FUNCTION_BLOCK ABSTRACT FB_PMLModuleBase IMPLEMENTS ITF_PMLModuleBase
VAR CONSTANT
	//Constant declarations
	PRODUCTION_DATA_ALARM_COUNT	: UDINT := 16;
END_VAR
VAR PERSISTENT
	//ITF_ProductionData internal variables
	tShiftLength: TIME := T#10M;
	nShiftProductionTarget	: DINT := 1000;
	fWarningMargin			: LREAL := 10;
	fProductionRate_Setpoint	: LREAL := 30;
	nRateAveragingCount		: DINT := 10;
END_VAR
VAR
	//ITF_PMLModuleBase internal property variables
	sAncestorIDs		: STRING;				//String concatenation of preceding parent IDs to prefix this module's ID
	bLogModeChanges 	: BOOL := TRUE; 		//Toggle to permit or suppress state change logging (Should be tied to HMI setting to optionally reduce event logger clutter)
	bLogStateChanges 	: BOOL := FALSE; 		//Toggle to permit or suppress state change logging (Should be tied to HMI setting to optionally reduce event logger clutter)
	nModuleID			: UDINT;					//Unique identifying number for the module
	sModuleName			: STRING;				//Human-readable module name for user-side messaging
	bEnabled			: BOOL := TRUE;			//Enables or disables the packml Machine of the module (prevents the module from going past idle)
	eModeCommand		: E_PMLUnitMode; 				//Current Commanded UnitMode of the module
	eStateCommand		: Tc3_PackML_V2.E_PMLCommand;
	eMode				: E_PMLUnitMode;		//Current UnitMode of the module
	eState				: Tc3_PackML_V2.E_PMLState;
	iMasterDataStructure_Adder : ITF_Tree_IndexBased;
	eCurrentAlarmSeverity		: TcEventSeverity;
	a_eParentFaultResponseDefinitions		: ARRAY[0..4] OF E_AlarmResponse := [	E_AlarmResponse.NoResponse,
																					E_AlarmResponse.NoResponse,
																					E_AlarmResponse.NoResponse,
																					E_AlarmResponse.Abort_ImmediateError,
																					E_AlarmResponse.Abort_ImmediateError];
	
	fbFIFO							: FB_FIFO_ULINT_Array;
	a_fbProductionDataAlarms		: ARRAY[1..PRODUCTION_DATA_ALARM_COUNT] OF FB_TcAlarm;
	fTemp : LREAL;



	//Communication Variables
	stPMLModuleBaseHMI	: ST_PMLModuleBase_HMI;		//Handles status and control communications with the HMI
	stPMLModuleBaseVISU	: ST_PMLModuleBase_VISU;	//Handles status and control communications with Visualizations
	fbExternalControl	: FB_ModuleExternalCommandControl;	//Handles commands from HMI/VISUS ^^ kind of overlaps with the structures above - TODO: Improve

	//Administration and Configuration Variables
	bInitialized 					: BOOL;					//TRUE when initialization code of the object is complete
	sID_Name						: STRING;				//"Module XX - 'Module Name' " Alarm and message utility phrase based off of nMachine ID and sMachineName
	
	//State and Mode control blocks
	fbModeManager 					: PML_UnitModeManager; 	//Manages operating mode transitions and rules
	fbStateMachine 					: PML_StateMachine; 	//Manages PackML state transitions
	fbCustomModes 					: PML_UnitModeConfig;	//Used to define custom machine modes if desired

	//State and Mode Status and Command variables
	sState							: STRING; 				//String representation of the current state
	eLastState						: E_PMLState;			//Last cycle PackML state
	eLastStateCommand				: E_PMLCommand;			//Previous received PackML state command
	eLastMode		 				: DINT;					//Last PackML mode 
	eLastModeCommand 				: E_PMLUnitMode;					//Previous received PackML mode command
	bStateTasksComplete				: BOOL := FALSE;					//All tasks to be performed at this program level are complete
	bNoStateTasksToComplete			: BOOL := TRUE;					//Indicates whether this stateneeds to perform tasks other than commanding its children
	bSubModulesReady				: BOOL;					//All submodules have reached the commanded state
	
	//Alarming and Logging variables - Some may or may not be necessary depending on final alarm system implementation ----------------------------------------------
	//These are for the newer TMC Excel import style alarm system
	a_fbPMLAlarms					: ARRAY[1..48] OF FB_TcAlarm;	//Array of alarms for PackML state and mode changes that exist in any PackML enabled module
	a_fbBaseAlarms					: ARRAY[1..32] OF FB_TcAlarm;		//Array of alarms for general module Alarms				
	fbPMLStateLogger				: FB_PMLStateLogger;				//Logs PackML state changes
	fbPMLModeLogger					: FB_PMLModeLogger;					//Logs PackML Mode changes

	// Alarm handling
	bActiveAlarm					: BOOL;					//module has an active alarm		TODO: Implement			
	bGlobalSafetyStatus				: BOOL;
	//********************************************************************************************************************
	// Sub Module variables
	// Used mostly for EMs and Machines, but ok for CM. They are just null	
	a_ITF_PackMLBase				: ARRAY[1..MAX_NO_OF_SUBMODULES] OF ITF_PMLModuleBase;	
	// Array of the PML sub unit info array used by the statemachine
	a_stPMLSubUnitInfo				: ARRAY[1..MAX_NO_OF_SUBMODULES] OF ST_PMLSubUnitInfo;
	nNumberOfSubModules				: UDINT := 0;	//calculated number of instantiated sub modules
	// This is the information for each module's submodules.
	PMLSubUnitInfoRef				: ST_PMLSubUnitInfoRef;				// Reference to the subunit information, used by the state machine
	//********************************************************************************************************************
	
	//Component variables - Allow iterative control of child components (Mostly used with Control Modules, but usable anywhere)
	a_ITF_Components				: ARRAY[1..MAX_NO_OF_COMPONENTS] OF ITF_ComponentBase;
	nNumberOfComponents				: UDINT := 0;	//calculated number of instantiated components
	
	//Miscellaneous Variables
	fLastProductionRate_Setpoint 	: LREAL;
	nIndex							: UDINT;		//Generic iteration value
	bSimulateAllChildren			: BOOL;
	a_sModeNames					: ARRAY[0..31] OF STRING;
	varInfo							: __SYSTEM.VAR_INFO;
	bReachedInitialDefaultStateAndMode	: BOOL;		//Toggles TRUE once a module has reached the default state and mode after startup, used to mute certain alarms during startup
	i: UDINT;
END_VAR

//*********************************************************
// !!!!! Code implementation only in CyclicLogic() method !!!!! 
//*********************************************************

METHOD Aborted
//*************************************************************************************************************************************************************************
//If you are about to write application specific code, note that any such code should exist within the "Application" directory using a Function Block that 'EXTENDS' this base Function Block!
//This particular method's functionality can be overriden in the extended block by creating a method of the same name, with desired functionality therein
//If the functionality of this base module is to be retained, but more functionality is desired, the extended method can contain a SUPER^.ThisMethodName(); call, which will call this code
//*************************************************************************************************************************************************************************

;
END_METHOD

METHOD AbortImmediate : BOOL
VAR_INPUT
END_VAR
eStateCommand := E_PMLCommand.ePMLCommand_Abort;
END_METHOD

METHOD AbortImmediateError : BOOL
VAR_INPUT
	sName		: STRING;
	bIsModule	: BOOL;
END_VAR
IF bIsModule THEN
	IF NOT a_fbBaseAlarms[E_BaseAlarms.SubModuleError].bRaised THEN
		F_RaiseAlarmWithStringParameters(a_fbBaseAlarms[E_BaseAlarms.SubModuleError],sModuleName,sName,'');
	END_IF
ELSE
	IF NOT a_fbBaseAlarms[E_BaseAlarms.ComponentError].bRaised THEN
		F_RaiseAlarmWithStringParameters(a_fbBaseAlarms[E_BaseAlarms.ComponentError],sModuleName,sName,'');
	END_IF
END_IF


eStateCommand := E_PMLCommand.ePMLCommand_Abort;
END_METHOD

METHOD Aborting
//*************************************************************************************************************************************************************************
//If you are about to write application specific code, note that any such code should exist within the "Application" directory using a Function Block that 'EXTENDS' this base Function Block!
//This particular method's functionality can be overriden in the extended block by creating a method of the same name, with desired functionality therein
//If the functionality of this base module is to be retained, but more functionality is desired, the extended method can contain a SUPER^.ThisMethodName(); call, which will call this code
//*************************************************************************************************************************************************************************

//Perform State tasks here
// Send abort command to all sub modules
FOR nIndex := 1 TO nNumberOfSubModules DO
	a_ITF_PackMLBase[nIndex].StateCommand:=ePMLCommand_Abort;
END_FOR

// All subunits in requested state?
bSubModulesReady := TRUE;

FOR nIndex := 1 TO nNumberOfSubModules DO
	bSubModulesReady := bSubModulesReady AND (a_ITF_PackMLBase[nIndex].State = ePMLState_Aborted);
END_FOR
IF bSubModulesReady AND (bStateTasksComplete OR bNoStateTasksToComplete) THEN
	bNoStateTasksToComplete := TRUE;
	bStateTasksComplete := FALSE;
	StateComplete();
END_IF
END_METHOD

METHOD AllowHMIControl : BOOL
VAR_INPUT
	bModuleOnly		: BOOL;	//If TRUE, only the PML module itself is controllable, If FALSE, all components become controllable as well
END_VAR
stPMLModuleBaseHMI.bHMIControlAvailable := TRUE;

IF bModuleOnly THEN
	FOR i := 1 TO nNumberOfComponents DO
		a_ITF_Components[i].BlockHMIControl();
	END_FOR
ELSE
	FOR i := 1 TO nNumberOfComponents DO
		a_ITF_Components[i].AllowHMIControl();
	END_FOR
END_IF
END_METHOD

PROPERTY AncestorIDs : STRING
GET
AncestorIDs := sAncestorIDs;
END_GET
SET
sAncestorIDs := AncestorIDs;
END_SET
END_PROPERTY

METHOD BlockHMIControl : BOOL
VAR_INPUT
END_VAR
stPMLModuleBaseHMI.bHMIControlAvailable := FALSE;

FOR i := 1 TO nNumberOfComponents DO
	a_ITF_Components[i].BlockHMIControl();
END_FOR
END_METHOD

METHOD Clearing
//*************************************************************************************************************************************************************************
//If you are about to write application specific code, note that any such code should exist within the "Application" directory using a Function Block that 'EXTENDS' this base Function Block!
//This particular method's functionality can be overriden in the extended block by creating a method of the same name, with desired functionality therein
//If the functionality of this base module is to be retained, but more functionality is desired, the extended method can contain a SUPER^.ThisMethodName(); call, which will call this code
//*************************************************************************************************************************************************************************

//Perform State tasks here
// Send clear command to all sub modules
FOR nIndex := 1 TO nNumberOfSubModules DO	
	a_ITF_PackMLBase[nIndex].StateCommand := ePMLCommand_Clear;
END_FOR

IF a_fbBaseAlarms[E_BaseAlarms.ComponentError].bRaised THEN
	a_fbBaseAlarms[E_BaseAlarms.ComponentError].Clear(0,0);
END_IF;

IF a_fbBaseAlarms[E_BaseAlarms.SubModuleError].bRaised THEN
	a_fbBaseAlarms[E_BaseAlarms.SubModuleError].Clear(0,0);
END_IF;


// All subunits in requested state?
bSubModulesReady	:= TRUE;
FOR nIndex:=1 TO nNumberOfComponents DO
	IF a_ITF_Components[nIndex].Error THEN
		a_ITF_Components[nIndex].Reset();
	END_IF
END_FOR

FOR nIndex:=1 TO nNumberOfComponents DO		
		bSubModulesReady := bSubModulesReady AND NOT a_ITF_Components[nIndex].Error;
END_FOR

FOR nIndex := 1 TO nNumberOfSubModules DO
	bSubModulesReady := bSubModulesReady AND (a_ITF_PackMLBase[nIndex].State = ePMLState_Stopped);
END_FOR
IF bSubModulesReady AND (bStateTasksComplete OR bNoStateTasksToComplete) THEN
	bNoStateTasksToComplete := TRUE;
	bStateTasksComplete := FALSE;
	StateComplete();
END_IF
END_METHOD

METHOD Complete
//*************************************************************************************************************************************************************************
//If you are about to write application specific code, note that any such code should exist within the "Application" directory using a Function Block that 'EXTENDS' this base Function Block!
//This particular method's functionality can be overriden in the extended block by creating a method of the same name, with desired functionality therein
//If the functionality of this base module is to be retained, but more functionality is desired, the extended method can contain a SUPER^.ThisMethodName(); call, which will call this code
//*************************************************************************************************************************************************************************

;
END_METHOD

METHOD Completing
//*************************************************************************************************************************************************************************
//If you are about to write application specific code, note that any such code should exist within the "Application" directory using a Function Block that 'EXTENDS' this base Function Block!
//This particular method's functionality can be overriden in the extended block by creating a method of the same name, with desired functionality therein
//If the functionality of this base module is to be retained, but more functionality is desired, the extended method can contain a SUPER^.ThisMethodName(); call, which will call this code
//*************************************************************************************************************************************************************************

//Perform State tasks here
// Send complete command to all sub modules
FOR nIndex := 1 TO nNumberOfSubModules DO
	a_ITF_PackMLBase[nIndex].StateCommand:=ePMLCommand_Complete;
END_FOR

// All subunits in requested state?
bSubModulesReady	:= TRUE;
FOR nIndex := 1 TO nNumberOfSubModules DO
	bSubModulesReady := bSubModulesReady AND (a_ITF_PackMLBase[nIndex].State = ePMLState_Complete);
END_FOR
IF bSubModulesReady AND (bStateTasksComplete OR bNoStateTasksToComplete) THEN
	bNoStateTasksToComplete := TRUE;
	bStateTasksComplete := FALSE;
	StateComplete();
END_IF
END_METHOD

METHOD ComponentMonitor : BOOL
VAR
	a_eAlarmResponses		: ARRAY[0..4] OF E_AlarmResponse;	//Temporary response array
END_VAR
FOR i:=1 TO nNumberOfComponents DO
	IF bSimulateAllChildren THEN
		a_ITF_Components[i].Simulate := TRUE;
	ELSE 
		a_ITF_Components[i].Simulate := FALSE;
	END_IF
	
	IF eMode = E_PMLUnitMode.ePMLUnitMode_Production THEN
		IF 		eState <> E_PMLState.ePMLState_Aborted
			AND eState <> E_PMLState.ePMLState_Aborting
			AND eState <> E_PMLState.ePMLState_Clearing
			AND eState <> E_PMLState.ePMLState_Stopped
			AND eState <> E_PMLState.ePMLState_Stopping
		THEN
			a_eAlarmResponses := a_ITF_Components[i].ParentResponseDefinitions;
			CASE a_eAlarmResponses[a_ITF_Components[i].CurrentAlarmSeverity] OF
				E_AlarmResponse.Abort_ImmediateError:
					AbortImmediateError(a_ITF_Components[i].Name, FALSE);
				E_AlarmResponse.Abort_Immediate:
					AbortImmediate();
				E_AlarmResponse.Stop_Immediate:
					StopImmediate();
				E_AlarmResponse.Stop_Controlled:
					StopControlled();
				E_AlarmResponse.Hold_Immediate:
					HoldImmediate();
				E_AlarmResponse.Suspend_Immediate:
					SuspendImmediate();
				E_AlarmResponse.Suspend_Controlled:
					SuspendControlled();
				E_AlarmResponse.NoResponse:
					;
			END_CASE
		ELSIF eState = E_PMLState.ePMLState_Stopped
			OR eState = E_PMLState.ePMLState_Stopping 
		THEN
			a_eAlarmResponses := a_ITF_Components[i].ParentResponseDefinitions;
			CASE a_eAlarmResponses[a_ITF_Components[i].CurrentAlarmSeverity] OF
				E_AlarmResponse.Abort_ImmediateError:
					AbortImmediateError(a_ITF_Components[i].Name, FALSE);
				E_AlarmResponse.Abort_Immediate:
					AbortImmediate();
				E_AlarmResponse.NoResponse:
					;
			END_CASE				
		END_IF
	END_IF		
END_FOR
END_METHOD

{attribute 'call_after_online_change_slot' := '<slot>'}
METHOD CreateEvents : BOOL
VAR_INPUT
END_VAR

VAR
END_VAR

F_CreateAllEventsInClass(	p_aAlarms := a_fbPMLAlarms,
							nClassSize := SIZEOF(TC_EVENTS.PMLAlarms),
							pInitEvent := ADR(TC_EVENTS.PMLAlarms.InitReferenceEvent),
							sPrefix := sID_Name);
							
F_CreateAllEventsInClass(	p_aAlarms := a_fbBaseAlarms,
							nClassSize := SIZEOF(TC_EVENTS.BaseAlarms),
							pInitEvent := ADR(TC_EVENTS.BaseAlarms.InitReferenceEvent),
							sPrefix := sID_Name);							
							
F_CreateAllEventsInClass(	p_aAlarms := a_fbProductionDataAlarms,
							nClassSize := SIZEOF(TC_EVENTS.ProductionData),
							pInitEvent := ADR(TC_EVENTS.ProductionData.InitReferenceEvent),
							sPrefix := sID_Name);
END_METHOD

PROPERTY CurrentAlarmSeverity : TcEventSeverity
GET
CurrentAlarmSeverity := eCurrentAlarmSeverity;
END_GET
END_PROPERTY

// 
// Cyclic Code
METHOD CyclicLogic
//*********************************************************
//If you are about to write actual machine implementation code, note that implementation code should exist within an implementation machine module block that extends this machine module base!
//*********************************************************

// First loop initialization code is triggered by highest level class
IF NOT bInitialized THEN			//Force initialization code of the object
	initialize();
	bInitialized := TRUE;
END_IF

//TODO: Condition state based on DEFAULT constant, right now it is a command, so a case statement translation to state would be necessary
IF NOT bReachedInitialDefaultStateAndMode AND eState = E_PMLState.ePMLState_Aborted AND eMode = ePMLUNITMODEDEFAULT THEN
	bReachedInitialDefaultStateAndMode := TRUE;
END_IF

//  call the subunits
FOR i := 1 TO nNumberOfSubModules DO	
	a_ITF_PackMLBase[i].CyclicLogic();								//Call the main cyclic loop of the subunits 
	a_stPMLSubUnitInfo[i].eState := a_ITF_PackMLBase[i].State;  	//Reflect the state of the subunits to the state machine of the module
END_FOR

FOR i:=1 TO nNumberOfComponents DO
	IF a_ITF_Components[i] <> 0 THEN
		a_ITF_Components[i].CyclicLogic();
	END_IF
END_FOR


// Mode control loop of the module
ModeControl();

// State control loop of the module
StateControl();

HMICommunication();
VISUCommunication();
fbExternalControl();
SubModuleMonitor();
ComponentMonitor();
HMIPermissions();

eCurrentAlarmSeverity := TcEventSeverity.Verbose;

eCurrentAlarmSeverity := F_GetMaxSeverityRaised(	a_fbAlarms := a_fbPMLAlarms,
													eCurrentSeverity := eCurrentAlarmSeverity);
eCurrentAlarmSeverity := F_GetMaxSeverityRaised(	a_fbAlarms := a_fbBaseAlarms,
													eCurrentSeverity := eCurrentAlarmSeverity);
END_METHOD

PROPERTY Enabled : BOOL
GET
Enabled := bEnabled;
END_GET
SET
bEnabled := Enabled;
END_SET
END_PROPERTY

METHOD Execute
//*************************************************************************************************************************************************************************
//If you are about to write application specific code, note that any such code should exist within the "Application" directory using a Function Block that 'EXTENDS' this base Function Block!
//This particular method's functionality can be overriden in the extended block by creating a method of the same name, with desired functionality therein
//If the functionality of this base module is to be retained, but more functionality is desired, the extended method can contain a SUPER^.ThisMethodName(); call, which will call this code
//*************************************************************************************************************************************************************************

;
END_METHOD

METHOD Held
//*************************************************************************************************************************************************************************
//If you are about to write application specific code, note that any such code should exist within the "Application" directory using a Function Block that 'EXTENDS' this base Function Block!
//This particular method's functionality can be overriden in the extended block by creating a method of the same name, with desired functionality therein
//If the functionality of this base module is to be retained, but more functionality is desired, the extended method can contain a SUPER^.ThisMethodName(); call, which will call this code
//*************************************************************************************************************************************************************************
END_METHOD

METHOD HMICommunication : BOOL
//Extend this method in extended FBs to communicate specific implementation data

//Process HMI requests
IF stPMLModuleBaseHMI.bIncomingHMIRequest AND NOT stPMLModuleBaseHMI.bHMICommandConfirmation THEN		//If a request has been issued by the HMI, and a previous request has not just E_SequenceState.Finished being processed
	
	IF stPMLModuleBaseHMI.bHMIControlAvailable THEN		//If the current conditions permit HMI control (Should be determined by the extended application components)
		IF stPMLModuleBaseHMI.bEnableHMIRequest THEN
			bEnabled := TRUE;
			stPMLModuleBaseHMI.bHMICommandConfirmation := TRUE;	//Confirm that the request has been processed
		END_IF
		IF stPMLModuleBaseHMI.bDisableHMIRequest THEN
			bEnabled := FALSE;
			stPMLModuleBaseHMI.bHMICommandConfirmation := TRUE;	//Confirm that the request has been processed
		END_IF
		IF stPMLModuleBaseHMI.bStateCommandHMIRequest THEN
			eStateCommand := stPMLModuleBaseHMI.eStateCommandHMIValue;
			//fbExternalControl.ExternalControlHMI.StateCommand := stPMLModuleBaseHMI.eStateCommandHMIValue;
			//fbExternalControl.ExternalControlHMI.StateCommandPulse := TRUE;
			stPMLModuleBaseHMI.bHMICommandConfirmation := TRUE;	//Confirm that the request has been processed
		END_IF
		IF stPMLModuleBaseHMI.bModeCommandHMIRequest THEN
			eModeCommand := stPMLModuleBaseHMI.eModeCommandHMIValue;
			//fbExternalControl.ExternalControlHMI.ModeCommand := stPMLModuleBaseHMI.eModeCommandHMIValue;
			//fbExternalControl.ExternalControlHMI.ModeCommandPulse := TRUE;
			stPMLModuleBaseHMI.bHMICommandConfirmation := TRUE;	//Confirm that the request has been processed
		END_IF
	END_IF
	
		//The following commands are always permissible, and are therefore not conditioned with bHMIControlAvailable
	IF stPMLModuleBaseHMI.bActivateStateLogHMIRequest THEN
		bLogStateChanges := TRUE;
		stPMLModuleBaseHMI.bHMICommandConfirmation := TRUE;	//Confirm that the request has been processed
	END_IF
	IF stPMLModuleBaseHMI.bDeactivateStateLogHMIRequest THEN
		bLogStateChanges := FALSE;
		stPMLModuleBaseHMI.bHMICommandConfirmation := TRUE;	//Confirm that the request has been processed
	END_IF
	IF stPMLModuleBaseHMI.bActivateModeLogHMIRequest THEN
		bLogModeChanges := TRUE;
		stPMLModuleBaseHMI.bHMICommandConfirmation := TRUE;	//Confirm that the request has been processed
	END_IF
	IF stPMLModuleBaseHMI.bDeactivateModeLogHMIRequest THEN
		bLogModeChanges := FALSE;
		stPMLModuleBaseHMI.bHMICommandConfirmation := TRUE;	//Confirm that the request has been processed
	END_IF		
END_IF


//Update HMI status info
stPMLModuleBaseHMI.bEnabled := bEnabled;
stPMLModuleBaseHMI.eMode := eMode;		//KAB eMode;
stPMLModuleBaseHMI.nModuleID := nModuleID;
stPMLModuleBaseHMI.sModuleName := sModuleName;
stPMLModuleBaseHMI.eState := eState;	//KAB eState;
stPMLModuleBaseHMI.bLogStateChanges := bLogStateChanges;
stPMLModuleBaseHMI.bLogModeChanges := bLogModeChanges;
stPMLModuleBaseHMI.a_sModeNames := a_sModeNames;
END_METHOD

PROPERTY HMIControlAvailable : BOOL
GET
HMIControlAvailable := stPMLModuleBaseHMI.bHMIControlAvailable;
END_GET
SET
stPMLModuleBaseHMI.bHMIControlAvailable := HMIControlAvailable;
END_SET
END_PROPERTY

METHOD HMIPermissions : BOOL
VAR_INPUT
END_VAR
//General Mode Based Monitoring and handling of HMI control
CASE eMode OF
//	====================================================================================================================================	
	E_PMLUnitMode.ePMLUnitMode_Production:			//=================================PRODUCTION MODE==================================
		CASE eState OF
			E_PMLState.ePMLState_Stopped:
				AllowHMIControl(bModuleOnly := TRUE);		//Allow control for recovery
			E_PMLState.ePMLState_Idle:
				BlockHMIControl();
			E_PMLState.ePMLState_Suspended:
				BlockHMIControl();
			E_PMLState.ePMLState_Execute:
				BlockHMIControl();
			E_PMLState.ePMLState_Aborted:
				AllowHMIControl(bModuleOnly := TRUE);		//Allow control for recovery
			E_PMLState.ePMLState_Held:
				AllowHMIControl(bModuleOnly := TRUE);		//Allow control for recovery
			E_PMLState.ePMLState_Complete:
				BlockHMIControl();
		END_CASE
		
//	====================================================================================================================================	
	E_PMLUnitMode.ePMLUnitMode_Manual:				//=================================MANUAL MODE======================================
		AllowHMIControl(bModuleOnly := FALSE);
//	====================================================================================================================================	
	E_PMLUnitMode.ePMLUnitMode_Maintenance:			//=================================MAINTENANCE MODE=================================
		AllowHMIControl(bModuleOnly := FALSE);	
END_CASE
END_METHOD

METHOD HoldControlled : BOOL
VAR_INPUT
END_VAR
END_METHOD

METHOD HoldImmediate : BOOL
VAR_INPUT
END_VAR
END_METHOD

METHOD Holding
//*************************************************************************************************************************************************************************
//If you are about to write application specific code, note that any such code should exist within the "Application" directory using a Function Block that 'EXTENDS' this base Function Block!
//This particular method's functionality can be overriden in the extended block by creating a method of the same name, with desired functionality therein
//If the functionality of this base module is to be retained, but more functionality is desired, the extended method can contain a SUPER^.ThisMethodName(); call, which will call this code
//*************************************************************************************************************************************************************************

//Perform State tasks here
// Send hold command to all sub modules
FOR nIndex := 1 TO nNumberOfSubModules DO
	a_ITF_PackMLBase[nIndex].StateCommand:=ePMLCommand_Hold;
END_FOR

// All subunits in requested state?
bSubModulesReady	:= TRUE;
FOR nIndex := 1 TO nNumberOfSubModules DO
	bSubModulesReady := bSubModulesReady AND (a_ITF_PackMLBase[nIndex].State = ePMLState_Held);
END_FOR
IF bSubModulesReady AND (bStateTasksComplete OR bNoStateTasksToComplete) THEN
	bNoStateTasksToComplete := TRUE;
	bStateTasksComplete := FALSE;
	StateComplete();
END_IF
END_METHOD

METHOD Idle
//*************************************************************************************************************************************************************************
//If you are about to write application specific code, note that any such code should exist within the "Application" directory using a Function Block that 'EXTENDS' this base Function Block!
//This particular method's functionality can be overriden in the extended block by creating a method of the same name, with desired functionality therein
//If the functionality of this base module is to be retained, but more functionality is desired, the extended method can contain a SUPER^.ThisMethodName(); call, which will call this code
//*************************************************************************************************************************************************************************
END_METHOD

METHOD initialize
VAR
	i : UDINT;
END_VAR
sID_Name := CONCAT(CONCAT(CONCAT(CONCAT(CONCAT('Module ', sAncestorIDs), UDINT_TO_STRING(nModuleID)), ' - '), sModuleName), ' '); 	//Creates a utility string for alarms and other messaging that reads (example text) - "Module 10 - Main Casepacker" to be followed by the alarm or message info
CreateEvents();

// Figure out how many Submodules were instantiated - they should be from 1 to X and not skip any indices.
nNumberOfSubModules := 0;
FOR i:=1 TO MAX_NO_OF_SUBMODULES DO
	IF a_ITF_PackMLBase[i] <> 0 THEN
		IF iMasterDataStructure_Adder <> 0 THEN
			iMasterDataStructure_Adder.AddNodeAsChildByName(sNewName := a_ITF_PackMLBase[i].ModuleName, sParentName := ModuleName);
		ELSIF NOT a_fbBaseAlarms[E_BaseAlarms.InvalidInterface].bRaised THEN
			varInfo :=  __VARINFO(iMasterDataStructure_Adder);
			F_RaiseAlarmWithStringParameters(a_fbBaseAlarms[E_BaseAlarms.InvalidInterface], sModuleName, varInfo.Symbol, '');	
		END_IF
		nNumberOfSubModules:=nNumberOfSubModules+1;
		
		a_ITF_PackMLBase[i].AncestorIDs := CONCAT(CONCAT(AncestorIDs, DINT_TO_STRING(ModuleID)), '_');
		a_ITF_PackMLBase[i].MasterDataStructure_Adder 	:= iMasterDataStructure_Adder;
		IF a_ITF_PackMLBase[i].ModuleID = 0 THEN	//If the ID was not manually initialized to anything at declaration, automatically assign it an ID
			a_ITF_PackMLBase[i].ModuleID := i;
		END_IF
	END_IF
END_FOR

nNumberOfComponents := 0;
FOR i:=1 TO MAX_NO_OF_COMPONENTS DO
	IF a_ITF_Components[i] <> 0 THEN

		a_ITF_Components[i].Name := CONCAT(CONCAT(sModuleName,' '),a_ITF_Components[i].Name);	//Add the name of the module as a prefix to the name given in the declaration initialization
		
		IF iMasterDataStructure_Adder <> 0 THEN
			iMasterDataStructure_Adder.AddNodeAsChildByName(sNewName := a_ITF_Components[i].Name, sParentName := ModuleName);
		ELSIF NOT a_fbBaseAlarms[E_BaseAlarms.InvalidInterface].bRaised THEN
			varInfo :=  __VARINFO(iMasterDataStructure_Adder);
			F_RaiseAlarmWithStringParameters(a_fbBaseAlarms[E_BaseAlarms.InvalidInterface], sModuleName, varInfo.Symbol, '');	
		END_IF
		nNumberOfComponents:=nNumberOfComponents+1;
	END_IF
END_FOR

fbExternalControl.Module := THIS^;

// <BASIC INITIALIZATION CODE, DO NOT CHANGE>
// Initialize subunit overview used by state machine
PMLSubUnitInfoRef.ArraySize := SIZEOF(a_stPMLSubUnitInfo);
PMLSubUnitInfoRef.NoOfSubUnits := nNumberOfSubModules;
PMLSubUnitInfoRef.pArray := ADR(a_stPMLSubUnitInfo);
// Point the state machine to the locally defined subunit info 
//fbStateMachine.stSubUnitInfoRef := PMLSubUnitInfoRef;
// <\BASIC INITIALIZATION CODE, DO NOT CHANGE>

// Activate all subunits by default, or change accordingly
FOR i:=1 TO nNumberOfSubModules DO
	a_stPMLSubUnitInfo[i].Active	:= TRUE;					// Follows Main State Machine
END_FOR

FOR i:=1 TO nNumberOfComponents DO
	IF a_ITF_Components[i] <> 0 THEN
		a_ITF_Components[i].Enabled := TRUE;
	END_IF
END_FOR
END_METHOD

PROPERTY LogModeChanges : BOOL
GET
LogModeChanges:= bLogModeChanges;
END_GET
SET
bLogModeChanges := LogModeChanges;
END_SET
END_PROPERTY

PROPERTY LogStateChanges : BOOL
GET
LogStateChanges:= bLogStateChanges;
END_GET
SET
bLogStateChanges := LogStateChanges;
END_SET
END_PROPERTY

PROPERTY MasterDataStructure_Adder :  ITF_Tree_IndexBased
GET
MasterDataStructure_Adder := iMasterDataStructure_Adder;
END_GET
SET
iMasterDataStructure_Adder := MasterDataStructure_Adder;
END_SET
END_PROPERTY

PROPERTY Mode : E_PMLUnitMode
GET
Mode := eMode;
END_GET
END_PROPERTY

PROPERTY ModeCommand : DINT
SET
eModeCommand := ModeCommand;
END_SET
END_PROPERTY

METHOD PRIVATE ModeControl
VAR
	i					: UDINT;
END_VAR
//On startup, Mode is invalid, set it to production
IF eMode = E_PMLUnitMode.ePMLUnitMode_Invalid 		THEN 
	fbModeManager.bExecute 		:= TRUE; 
	eModeCommand			 	:= ePMLUNITMODEDEFAULT; 
	eLastModeCommand 			:= eModeCommand;
//If mode is valid and the command has changed, attempt to change modes
ELSIF eModeCommand <> eLastModeCommand 					THEN
	//DONKEY : logging to be implemented
	fbModeManager.bExecute 		:= TRUE;
	eLastModeCommand 			:= eModeCommand;
END_IF

//Handles mode changes based on eModeCommand and the state transition rules defined in the pre-defined protected modes or custom modes
fbModeManager(
	eModeCommand			:= eModeCommand, 
	eState					:= eState, 			
	eModeStatus				=> eMode, 
	bDone					=> , 
	bError					=> , 
	nErrorId				=> 
	);
	
IF fbModeManager.bError AND bReachedInitialDefaultStateAndMode THEN
	IF NOT a_fbPMLAlarms[E_PMLAlarms.ModeCommandInvalid].bRaised THEN
		a_fbPMLAlarms[E_PMLAlarms.ModeCommandInvalid].Raise(0);
	END_IF
ELSIF a_fbPMLAlarms[E_PMLAlarms.ModeCommandInvalid].bRaised THEN
	a_fbPMLAlarms[E_PMLAlarms.ModeCommandInvalid].Clear(0,0);
END_IF

// Reset mode control command
fbModeManager.bExecute 		:= FALSE;

//If PackML mode has changed
IF fbModeManager.eModeStatus <> eLastMode  THEN 
	eLastMode := fbModeManager.eModeStatus; 
	//If state change logging is not suppressed
 	IF bLogModeChanges THEN 
		fbPMLModeLogger(
			a_fbPMLAlarms := a_fbPMLAlarms,
			sModulePrefix := sID_Name,
			Mode := fbModeManager.eModeStatus);	
	END_IF	
	// Change SubModules
	FOR i := 1 TO nNumberOfSubModules DO
		a_ITF_PackMLBase[i].ModeCommand := fbModeManager.eModeStatus;		//Call the SetMode loop of the subunits 
	END_FOR

END_IF
END_METHOD

PROPERTY ModuleID : UDINT
GET
ModuleID := nModuleID;
END_GET
SET
nModuleID := ModuleID;
END_SET
END_PROPERTY

PROPERTY ModuleName : STRING
GET
ModuleName := sModuleName;
END_GET
SET
sModuleName := ModuleName;
END_SET
END_PROPERTY

PROPERTY ParentResponse_Critical : E_AlarmResponse
GET
ParentResponse_Critical := a_eParentFaultResponseDefinitions[TcEventSeverity.Critical];
END_GET
SET
a_eParentFaultResponseDefinitions[TcEventSeverity.Critical] := ParentResponse_Critical;
END_SET
END_PROPERTY

PROPERTY ParentResponse_Error : E_AlarmResponse
GET
ParentResponse_Error := a_eParentFaultResponseDefinitions[TcEventSeverity.Error];
END_GET
SET
a_eParentFaultResponseDefinitions[TcEventSeverity.Error] := ParentResponse_Error;
END_SET
END_PROPERTY

PROPERTY ParentResponse_Warning : E_AlarmResponse
GET
ParentResponse_Warning := a_eParentFaultResponseDefinitions[TcEventSeverity.Warning];
END_GET
SET
a_eParentFaultResponseDefinitions[TcEventSeverity.Warning] := ParentResponse_Warning;
END_SET
END_PROPERTY

PROPERTY ParentResponseDef : ARRAY[0..4] OF E_AlarmResponse
GET
ParentResponseDef[TcEventSeverity.Verbose] := a_eParentFaultResponseDefinitions[TcEventSeverity.Verbose];
ParentResponseDef[TcEventSeverity.Info] := a_eParentFaultResponseDefinitions[TcEventSeverity.Info];
ParentResponseDef[TcEventSeverity.Warning] := a_eParentFaultResponseDefinitions[TcEventSeverity.Warning];
ParentResponseDef[TcEventSeverity.Error] := a_eParentFaultResponseDefinitions[TcEventSeverity.Error];
ParentResponseDef[TcEventSeverity.Critical] := a_eParentFaultResponseDefinitions[TcEventSeverity.Critical];
END_GET
SET
a_eParentFaultResponseDefinitions[TcEventSeverity.Verbose] := ParentResponseDef[TcEventSeverity.Verbose];
a_eParentFaultResponseDefinitions[TcEventSeverity.Info] := ParentResponseDef[TcEventSeverity.Info];
a_eParentFaultResponseDefinitions[TcEventSeverity.Warning] := ParentResponseDef[TcEventSeverity.Warning];
a_eParentFaultResponseDefinitions[TcEventSeverity.Error] := ParentResponseDef[TcEventSeverity.Error];
a_eParentFaultResponseDefinitions[TcEventSeverity.Critical] := ParentResponseDef[TcEventSeverity.Critical];
END_SET
END_PROPERTY

METHOD Resetting
//*************************************************************************************************************************************************************************
//If you are about to write application specific code, note that any such code should exist within the "Application" directory using a Function Block that 'EXTENDS' this base Function Block!
//This particular method's functionality can be overriden in the extended block by creating a method of the same name, with desired functionality therein
//If the functionality of this base module is to be retained, but more functionality is desired, the extended method can contain a SUPER^.ThisMethodName(); call, which will call this code
//*************************************************************************************************************************************************************************

//Perform State tasks here
// Send clear/reset command to all sub modules
//As long as this module is in the "Resetting" state, it will attempt to get all modules to Idle by sending abort, clear, and reset commands as appropriate to its children until they do
FOR nIndex := 1 TO nNumberOfSubModules DO
	IF a_ITF_PackMLBase[nIndex].State=ePMLState_Stopped OR a_ITF_PackMLBase[nIndex].State=ePMLState_Complete THEN
		a_ITF_PackMLBase[nIndex].StateCommand:=ePMLCommand_Reset;
	ELSIF a_ITF_PackMLBase[nIndex].State=ePMLState_Aborted THEN
		a_ITF_PackMLBase[nIndex].StateCommand:=ePMLCommand_Clear;
	ELSIF a_ITF_PackMLBase[nIndex].State=ePMLState_Clearing OR a_ITF_PackMLBase[nIndex].State=ePMLState_Stopping 
		OR a_ITF_PackMLBase[nIndex].State=ePMLState_Resetting OR a_ITF_PackMLBase[nIndex].State=ePMLState_Idle THEN
		;
	ELSE
		a_ITF_PackMLBase[nIndex].StateCommand:=ePMLCommand_Abort;
	END_IF
END_FOR

FOR nIndex:=1 TO nNumberOfComponents DO
	IF NOT a_ITF_Components[nIndex].Enabled THEN
		a_ITF_Components[nIndex].Enabled := TRUE;
	END_IF
END_FOR


// All subunits in requested state?
bSubModulesReady	:= TRUE;

FOR nIndex:=1 TO nNumberOfComponents DO		
	bSubModulesReady := bSubModulesReady AND a_ITF_Components[nIndex].Ready;
END_FOR

FOR nIndex := 1 TO nNumberOfSubModules DO
	bSubModulesReady := bSubModulesReady AND (a_ITF_PackMLBase[nIndex].State = ePMLState_Idle);
END_FOR
IF bSubModulesReady AND (bStateTasksComplete OR bNoStateTasksToComplete) THEN
	bNoStateTasksToComplete := TRUE;
	bStateTasksComplete := FALSE;
	StateComplete();
END_IF
END_METHOD

PROPERTY SimulateAllChildren : BOOL
GET
SimulateAllChildren := bSimulateAllChildren;
END_GET
SET
bSimulateAllChildren := SimulateAllChildren;
END_SET
END_PROPERTY

METHOD Starting
//*************************************************************************************************************************************************************************
//If you are about to write application specific code, note that any such code should exist within the "Application" directory using a Function Block that 'EXTENDS' this base Function Block!
//This particular method's functionality can be overriden in the extended block by creating a method of the same name, with desired functionality therein
//If the functionality of this base module is to be retained, but more functionality is desired, the extended method can contain a SUPER^.ThisMethodName(); call, which will call this code
//*************************************************************************************************************************************************************************

//Perform State tasks here
// Send start command to all sub modules
FOR nIndex := 1 TO nNumberOfSubModules DO
	a_ITF_PackMLBase[nIndex].StateCommand:=ePMLCommand_Start;
END_FOR

// All subunits in requested state?
bSubModulesReady	:= TRUE; 
FOR nIndex := 1 TO nNumberOfSubModules DO
	bSubModulesReady := bSubModulesReady AND (a_ITF_PackMLBase[nIndex].State = ePMLState_Execute);
END_FOR 
IF bSubModulesReady AND (bStateTasksComplete OR bNoStateTasksToComplete) THEN
	bNoStateTasksToComplete := TRUE;
	bStateTasksComplete := FALSE;
	StateComplete();
END_IF
END_METHOD

PROPERTY State : Tc3_PackML_V2.E_PMLState
GET
State := eState;
END_GET
END_PROPERTY

PROPERTY StateCommand : Tc3_PackML_V2.E_PMLCommand
SET
IF 	eMode <> E_PMLUnitMode.ePMLUnitMode_Invalid 	AND
 	eState <> E_PMLState.ePMLState_Undefined 			THEN 
	eStateCommand := StateCommand;
END_IF
END_SET
END_PROPERTY

METHOD StateComplete
//*************************************************************************************************************************************************************************
//If you are about to write application specific code, note that any such code should exist within the "Application" directory using a Function Block that 'EXTENDS' this base Function Block!
//This particular method's functionality can be overriden in the extended block by creating a method of the same name, with desired functionality therein
//If the functionality of this base module is to be retained, but more functionality is desired, the extended method can contain a SUPER^.ThisMethodName(); call, which will call this code
//*************************************************************************************************************************************************************************

fbStateMachine.M_StateComplete();
END_METHOD

METHOD PRIVATE StateControl
//On startup, state is invalid, set it to default
IF eState = E_PMLState.ePMLState_Undefined 				AND 
	eMode <> E_PMLUnitMode.ePMLUnitMode_Invalid 	THEN 
	eStateCommand 	:= ePMLSTATEDEFAULT; 
END_IF

//Call PackML state machine	
fbStateMachine(
	eMode				:= eMode, 
	eCommand			:= eStateCommand, 
	stSubUnitInfoRef	:= ,
	stOptions			:= , 
	eState				=> eState, 
	sState 				=> sState, 
	bError				=> , 
	nErrorID			=> );

//If PackML state has changed
IF eState <> eLastState  THEN 
	eLastState := eState; 
	bNoStateTasksToComplete := TRUE;
END_IF 
	
IF bReachedInitialDefaultStateAndMode THEN
	//Log appropriate state changes
	fbPMLStateLogger(
		a_fbPMLAlarms := a_fbPMLAlarms, 
		sModulePrefix := SID_Name, 
		eState := eState,
		bLogAllChanges := bLogStateChanges);	
END_IF

// Call appropriate method depending on current PackML state
CASE eState OF
	E_PMLState.ePMLState_Undefined:
		Undefined();
	E_PMLState.ePMLState_Clearing:
		Clearing();
	E_PMLState.ePMLState_Stopped:
		Stopped();
	E_PMLState.ePMLState_Starting:
		Starting();
	E_PMLState.ePMLState_Idle:
		Idle();
	E_PMLState.ePMLState_Suspended:
		Suspended();
	E_PMLState.ePMLState_Execute:
		Execute();
	E_PMLState.ePMLState_Stopping:
		Stopping();
	E_PMLState.ePMLState_Aborting:
		Aborting();
	E_PMLState.ePMLState_Aborted:
		Aborted();
	E_PMLState.ePMLState_Holding:
		Holding();
	E_PMLState.ePMLState_Held:
		Held();
	E_PMLState.ePMLState_Unholding:
		Unholding();
	E_PMLState.ePMLState_Suspending:
		Suspending();
	E_PMLState.ePMLState_Unsuspending:
		Unsuspending();
	E_PMLState.ePMLState_Resetting:   	
		Resetting();
	E_PMLState.ePMLState_Completing:
		Completing();
	E_PMLState.ePMLState_Complete:
		Complete();
END_CASE
END_METHOD

METHOD StopControlled : BOOL
VAR_INPUT
END_VAR
END_METHOD

METHOD StopImmediate : BOOL
VAR_INPUT
END_VAR
eStateCommand := E_PMLCommand.ePMLCommand_Stop;
END_METHOD

METHOD Stopped
//*************************************************************************************************************************************************************************
//If you are about to write application specific code, note that any such code should exist within the "Application" directory using a Function Block that 'EXTENDS' this base Function Block!
//This particular method's functionality can be overriden in the extended block by creating a method of the same name, with desired functionality therein
//If the functionality of this base module is to be retained, but more functionality is desired, the extended method can contain a SUPER^.ThisMethodName(); call, which will call this code
//*************************************************************************************************************************************************************************
END_METHOD

METHOD Stopping
//*************************************************************************************************************************************************************************
//If you are about to write application specific code, note that any such code should exist within the "Application" directory using a Function Block that 'EXTENDS' this base Function Block!
//This particular method's functionality can be overriden in the extended block by creating a method of the same name, with desired functionality therein
//If the functionality of this base module is to be retained, but more functionality is desired, the extended method can contain a SUPER^.ThisMethodName(); call, which will call this code
//*************************************************************************************************************************************************************************

//Perform State tasks here
// Send stop command to all sub modules
FOR nIndex := 1 TO nNumberOfSubModules DO
	a_ITF_PackMLBase[nIndex].StateCommand:=ePMLCommand_Stop;
END_FOR

// All subunits in requested state?
bSubModulesReady	:= TRUE;
FOR nIndex := 1 TO nNumberOfSubModules DO
	bSubModulesReady := bSubModulesReady AND (a_ITF_PackMLBase[nIndex].State = ePMLState_Stopped OR a_ITF_PackMLBase[nIndex].State = ePMLState_Aborted);
END_FOR
IF bSubModulesReady AND (bStateTasksComplete OR bNoStateTasksToComplete) THEN
	bNoStateTasksToComplete := TRUE;
	bStateTasksComplete := FALSE;
	StateComplete();
END_IF
END_METHOD

METHOD SubModuleMonitor : BOOL
VAR
	a_eAlarmResponses		: ARRAY[0..4] OF E_AlarmResponse;	//Temporary response array	
END_VAR

FOR i := 1 TO nNumberOfSubModules DO
	
	IF bSimulateAllChildren THEN
		a_ITF_PackMLBase[i].SimulateAllChildren := TRUE;
	ELSE
		a_ITF_PackMLBase[i].SimulateAllChildren := FALSE;
	END_IF

	
	IF eMode = E_PMLUnitMode.ePMLUnitMode_Production THEN		
		IF 		eState <> E_PMLState.ePMLState_Aborted
			AND eState <> E_PMLState.ePMLState_Aborting
			AND eState <> E_PMLState.ePMLState_Clearing
			AND eState <> E_PMLState.ePMLState_Stopped
			AND eState <> E_PMLState.ePMLState_Stopping
		THEN
			a_eAlarmResponses := a_ITF_PackMLBase[i].ParentResponseDef;
			CASE a_eAlarmResponses[a_ITF_PackMLBase[i].CurrentAlarmSeverity] OF
				E_AlarmResponse.Abort_ImmediateError:
					AbortImmediateError(a_ITF_PackMLBase[i].ModuleName, TRUE);
				E_AlarmResponse.Abort_Immediate:
					AbortImmediate();
				E_AlarmResponse.Stop_Immediate:
					StopImmediate();
				E_AlarmResponse.Stop_Controlled:
					StopControlled();
				E_AlarmResponse.Hold_Immediate:
					HoldImmediate();
				E_AlarmResponse.Suspend_Immediate:
					SuspendImmediate();
				E_AlarmResponse.Suspend_Controlled:
					SuspendControlled();
				E_AlarmResponse.NoResponse:
					;
			END_CASE
		ELSIF eState = E_PMLState.ePMLState_Stopped
			OR eState = E_PMLState.ePMLState_Stopping 
		THEN
			a_eAlarmResponses := a_ITF_PackMLBase[i].ParentResponseDef;
			CASE a_eAlarmResponses[a_ITF_PackMLBase[i].CurrentAlarmSeverity] OF
				E_AlarmResponse.Abort_ImmediateError:
					AbortImmediateError(a_ITF_PackMLBase[i].ModuleName, TRUE);
				E_AlarmResponse.Abort_Immediate:
					AbortImmediate();
				E_AlarmResponse.NoResponse:
					;
			END_CASE				
		END_IF
	END_IF
END_FOR
END_METHOD

METHOD SuspendControlled : BOOL
VAR_INPUT
END_VAR
END_METHOD

METHOD Suspended
//*************************************************************************************************************************************************************************
//If you are about to write application specific code, note that any such code should exist within the "Application" directory using a Function Block that 'EXTENDS' this base Function Block!
//This particular method's functionality can be overriden in the extended block by creating a method of the same name, with desired functionality therein
//If the functionality of this base module is to be retained, but more functionality is desired, the extended method can contain a SUPER^.ThisMethodName(); call, which will call this code
//*************************************************************************************************************************************************************************
END_METHOD

METHOD SuspendImmediate : BOOL
VAR_INPUT
END_VAR
END_METHOD

METHOD Suspending
//*************************************************************************************************************************************************************************
//If you are about to write application specific code, note that any such code should exist within the "Application" directory using a Function Block that 'EXTENDS' this base Function Block!
//This particular method's functionality can be overriden in the extended block by creating a method of the same name, with desired functionality therein
//If the functionality of this base module is to be retained, but more functionality is desired, the extended method can contain a SUPER^.ThisMethodName(); call, which will call this code
//*************************************************************************************************************************************************************************

//Perform State tasks here
// Send suspend command to all sub modules
FOR nIndex := 1 TO nNumberOfSubModules DO
	a_ITF_PackMLBase[nIndex].StateCommand:=ePMLCommand_Suspend;
END_FOR

// All subunits in requested state?
bSubModulesReady	:= TRUE;
FOR nIndex := 1 TO nNumberOfSubModules DO
	bSubModulesReady := bSubModulesReady AND (a_ITF_PackMLBase[nIndex].State = ePMLState_Suspended);
END_FOR
IF bSubModulesReady AND (bStateTasksComplete OR bNoStateTasksToComplete) THEN
	bNoStateTasksToComplete := TRUE;
	bStateTasksComplete := FALSE;
	StateComplete();
END_IF
END_METHOD

PROPERTY TargetProductionRate : LREAL
GET
TargetProductionRate := fProductionRate_Setpoint;
END_GET
SET
fProductionRate_Setpoint := TargetProductionRate;
END_SET
END_PROPERTY

METHOD Undefined
//*************************************************************************************************************************************************************************
//If you are about to write application specific code, note that any such code should exist within the "Application" directory using a Function Block that 'EXTENDS' this base Function Block!
//This particular method's functionality can be overriden in the extended block by creating a method of the same name, with desired functionality therein
//If the functionality of this base module is to be retained, but more functionality is desired, the extended method can contain a SUPER^.ThisMethodName(); call, which will call this code
//*************************************************************************************************************************************************************************
END_METHOD

METHOD Unholding
//*************************************************************************************************************************************************************************
//If you are about to write application specific code, note that any such code should exist within the "Application" directory using a Function Block that 'EXTENDS' this base Function Block!
//This particular method's functionality can be overriden in the extended block by creating a method of the same name, with desired functionality therein
//If the functionality of this base module is to be retained, but more functionality is desired, the extended method can contain a SUPER^.ThisMethodName(); call, which will call this code
//*************************************************************************************************************************************************************************

//Perform State tasks here
// Send unhold command to all sub modules
FOR nIndex := 1 TO nNumberOfSubModules DO
	a_ITF_PackMLBase[nIndex].StateCommand:=ePMLCommand_Unhold;
END_FOR

// All subunits in requested state?
bSubModulesReady	:= TRUE;
FOR nIndex := 1 TO nNumberOfSubModules DO
	bSubModulesReady := bSubModulesReady AND (a_ITF_PackMLBase[nIndex].State = ePMLState_Execute);
END_FOR
IF bSubModulesReady AND (bStateTasksComplete OR bNoStateTasksToComplete) THEN
	bNoStateTasksToComplete := TRUE;
	bStateTasksComplete := FALSE;
	StateComplete();
END_IF
END_METHOD

METHOD Unsuspending
//*************************************************************************************************************************************************************************
//If you are about to write application specific code, note that any such code should exist within the "Application" directory using a Function Block that 'EXTENDS' this base Function Block!
//This particular method's functionality can be overriden in the extended block by creating a method of the same name, with desired functionality therein
//If the functionality of this base module is to be retained, but more functionality is desired, the extended method can contain a SUPER^.ThisMethodName(); call, which will call this code
//*************************************************************************************************************************************************************************

//Perform State tasks here
// Send unsuspend command to all sub modules
FOR nIndex := 1 TO nNumberOfSubModules DO
	a_ITF_PackMLBase[nIndex].StateCommand:=ePMLCommand_Unsuspend;
END_FOR

// All subunits in requested state?
bSubModulesReady	:= TRUE;
FOR nIndex := 1 TO nNumberOfSubModules DO
	bSubModulesReady := bSubModulesReady AND (a_ITF_PackMLBase[nIndex].State = ePMLState_Execute);
END_FOR
IF bSubModulesReady AND (bStateTasksComplete OR bNoStateTasksToComplete) THEN
	bNoStateTasksToComplete := TRUE;
	bStateTasksComplete := FALSE;
	StateComplete();
END_IF
END_METHOD

METHOD VISUCommunication : BOOL
VAR_INPUT
END_VAR

fbExternalControl.ExternalControlVISU.ClearPressed := stPMLModuleBaseVISU.bClearPressed;
fbExternalControl.ExternalControlVISU.ResetPressed := stPMLModuleBaseVISU.bResetPressed;
fbExternalControl.ExternalControlVISU.StartPressed := stPMLModuleBaseVISU.bStartPressed;
fbExternalControl.ExternalControlVISU.StopPressed := stPMLModuleBaseVISU.bStopPressed;


//Update VISU status info
stPMLModuleBaseVISU.bEnabled := bEnabled;
stPMLModuleBaseVISU.eMode := eMode;		
stPMLModuleBaseVISU.nModuleID := nModuleID;
stPMLModuleBaseVISU.sModuleName := sModuleName;
stPMLModuleBaseVISU.eState := eState;	

// Mode logic here.  Only taking the button from the visualizations
IF stPMLModuleBaseVISU.bProductionPressed AND eMode <> E_PMLUnitMode.ePMLUnitMode_Production THEN
	fbExternalControl.ExternalControlVISU.ModeCommand := E_PMLUnitMode.ePMLUnitMode_Production;
	fbExternalControl.ExternalControlVISU.ModeCommandPulse := TRUE;
END_IF
IF stPMLModuleBaseVISU.bMaintenancePressed AND eMode <> E_PMLUnitMode.ePMLUnitMode_Maintenance THEN
	fbExternalControl.ExternalControlVISU.ModeCommand := E_PMLUnitMode.ePMLUnitMode_Maintenance;
	fbExternalControl.ExternalControlVISU.ModeCommandPulse := TRUE;
END_IF
IF stPMLModuleBaseVISU.bManualPressed AND eMode <> E_PMLUnitMode.ePMLUnitMode_Manual THEN
	fbExternalControl.ExternalControlVISU.ModeCommand := E_PMLUnitMode.ePMLUnitMode_Manual;
	fbExternalControl.ExternalControlVISU.ModeCommandPulse := TRUE;
END_IF

// Extra buttons from Visu here for state changes than the standard 4
// Abort
IF stPMLModuleBaseVISU.bAbortPressed THEN
	CASE eState OF
		ePMLState_Aborted,
		ePMLState_Aborting:
			// DO Nothing
	ELSE
		fbExternalControl.ExternalControlVISU.StateCommand := E_PMLCommand.ePMLCommand_Abort;
		fbExternalControl.ExternalControlVISU.StateCommandPulse := TRUE;	
	END_CASE
END_IF

// Hold
IF stPMLModuleBaseVISU.bHoldPressed THEN
	IF eState = ePMLState_Execute THEN
		fbExternalControl.ExternalControlVISU.StateCommand := E_PMLCommand.ePMLCommand_Hold;
		fbExternalControl.ExternalControlVISU.StateCommandPulse := TRUE;	
	END_IF
END_IF

// unHold
IF stPMLModuleBaseVISU.bUnholdPressed THEN
	IF eState = ePMLState_Held THEN
		fbExternalControl.ExternalControlVISU.StateCommand := E_PMLCommand.ePMLCommand_Unhold;
		fbExternalControl.ExternalControlVISU.StateCommandPulse := TRUE;	
	END_IF
END_IF

// Suspend
IF stPMLModuleBaseVISU.bSuspendPressed THEN
	IF eState = ePMLState_Execute THEN
		fbExternalControl.ExternalControlVISU.StateCommand := E_PMLCommand.ePMLCommand_Suspend;
		fbExternalControl.ExternalControlVISU.StateCommandPulse := TRUE;	
	END_IF
END_IF

// unSuspend
IF stPMLModuleBaseVISU.bUnsuspendPressed THEN
	IF eState = ePMLState_Suspended THEN
		fbExternalControl.ExternalControlVISU.StateCommand := E_PMLCommand.ePMLCommand_Unsuspend;
		fbExternalControl.ExternalControlVISU.StateCommandPulse := TRUE;	
	END_IF
END_IF
END_METHOD

END_FUNCTION_BLOCK

(* stored: Version 1.1.0.1, ProductVersion 3.1.4024.11
   POU FB_PMLModuleBase: Id {b51128fe-fac6-441f-bd13-bfcb90049779}, SpecialFunc None
   Folder 01_ITF_PMLModuleBase: Id {7853c128-7150-499f-afd2-1cc47b02c7fb}
   Folder 01_Properties: Id {3f6fcce0-20d1-42fa-8d51-cf636ece4a9f}
   Folder 01_Config: Id {ea82163c-dcb7-40a8-a188-494f28a69630}
   Folder 02_Control: Id {0f49fae0-d86c-4069-99a8-907b07387580}
   Folder 03_Status: Id {84ded71b-93ac-410b-9a46-f376b2f39afb}
   Folder 02_Methods: Id {a47a966b-0b31-4e95-a3f6-5bd2e7b2f305}
   Folder Methods: Id {2374c43a-8b69-4250-ac37-650855e4142c}
   Folder 01_TransitionStates: Id {2813ee04-f5e3-4130-bb47-4373fa697726}
   Folder 02_PrimaryStates: Id {fdb26b20-d68a-43a5-9170-8c0cae9f966b}
   Folder 03_Monitoring: Id {0990b033-a812-4275-8ada-e06b2ca591b8}
   Folder 04_HMI: Id {0a574e76-6dab-426e-9c46-435414520792}
   Folder 05_AlarmHandling: Id {ad4fcf9c-0649-4b81-962f-40ddfe173e03}
   Method Aborted: Id {f4c80f4a-1f00-40f6-a791-318ec4b3278d}
   Method AbortImmediate: Id {3e55effc-a31f-4c38-a8a8-79f762ad7483}
   Method AbortImmediateError: Id {0f7de373-7b18-4301-aa32-84fc879a215e}
   Method Aborting: Id {ff7d5dfb-dd97-4700-92b4-3318a8a33dc3}
   Method AllowHMIControl: Id {8101f876-b4c9-49ea-be68-caa3d7179c06}
   Property AncestorIDs: Id {e9e1bc49-319c-49cf-ab24-edd60fccd3be}
   Get Get: Id {0d53a6f0-66af-4585-b735-0971eb97a602}
   Set Set: Id {f5655c38-0ec4-46ea-a0ed-5b08ec4b6fbd}
   Method BlockHMIControl: Id {6644c279-6fd0-47e2-a8e9-51778ec50ccd}
   Method Clearing: Id {6112c2e2-beb3-4b32-8c5f-7d289837fbce}
   Method Complete: Id {be38325c-ec06-4d18-82f0-c5961644db83}
   Method Completing: Id {25f6dadc-f2af-4e8f-bc90-78652fde6245}
   Method ComponentMonitor: Id {8175b5fe-f316-43ef-bef8-f03aa4ce0b3d}
   Method CreateEvents: Id {6bbb8cab-407d-45ac-8da1-6eb5ce7199bf}
   Property CurrentAlarmSeverity: Id {60fa6b26-f46a-4896-b539-afba05ef03bc}
   Get Get: Id {99112b04-4f01-4857-b0c7-d9fee82ac72b}
   Method CyclicLogic: Id {71af2bab-1028-44ec-8e3b-3536f0513c8e}
   Property Enabled: Id {a21599c5-6ae5-44f0-9223-afd1d8212c97}
   Get Get: Id {a6e327b1-41a2-4dd3-a0f8-24a28f9d1b3a}
   Set Set: Id {c5f0beb9-4653-47d9-893f-db8a432ad5d6}
   Method Execute: Id {26a49972-0a12-441d-92db-f9f223493eea}
   Method Held: Id {70dc6f04-1202-4345-ae9f-cc19428dcb1a}
   Method HMICommunication: Id {0f3b5e33-30dd-42a6-9468-c84dc53cce4a}
   Property HMIControlAvailable: Id {52f6c443-837f-4981-bfb9-75a309035060}
   Get Get: Id {d77cfdae-241d-47d6-9a7d-0a2f337596b6}
   Set Set: Id {a4b129d9-36a6-4e6e-a4e9-6de05e71bc5b}
   Method HMIPermissions: Id {5b677aa7-4ac1-443a-a993-772808975d8a}
   Method HoldControlled: Id {34a57a82-a45f-4e9f-bfac-d3a59430bbc7}
   Method HoldImmediate: Id {4f135bf7-6681-48b2-8727-b043804f866e}
   Method Holding: Id {4c4a9600-833f-4e2c-8c49-79d528d4d25d}
   Method Idle: Id {b9ab53ad-9d66-4112-a551-29e98d9dd437}
   Method initialize: Id {ce22347d-434e-4e9b-a860-79a350477497}
   Property LogModeChanges: Id {021783ae-5efd-4506-a012-4d08fd7e83f7}
   Get Get: Id {5e483759-154e-4761-b62a-a7c816d2ebfc}
   Set Set: Id {f46d3f1b-f363-4efb-8060-ae4e55813e7e}
   Property LogStateChanges: Id {66903c14-00c7-433b-8055-be34247fabbb}
   Get Get: Id {e672ec04-4b20-4c25-8d8d-9f55944d549a}
   Set Set: Id {5c42da14-b508-4ff1-b2f1-616dcf8c8ef8}
   Property MasterDataStructure_Adder: Id {df8bfb91-605f-4717-a7ce-9c6f277783e2}
   Get Get: Id {3f3aa2d9-680a-40a0-8573-571382f13def}
   Set Set: Id {53ffe855-67b4-4cc8-89ce-cf214fc8217c}
   Property Mode: Id {bc2b045c-1313-4030-8d9b-1e43964fed78}
   Get Get: Id {1dd33fe5-9737-46ae-8efa-b652739a2309}
   Property ModeCommand: Id {581c69c3-be81-4fff-9cf6-24ab11c559c3}
   Set Set: Id {428042c2-2a29-4c07-9a8f-eebad7e0d1dc}
   Method ModeControl: Id {8251b72f-7e35-4652-98c5-3fb000f5552b}
   Property ModuleID: Id {09c9c517-9d6d-4453-9051-a5bffda96bf8}
   Get Get: Id {98b97e95-2030-4cdf-9c6a-02fd26d24c96}
   Set Set: Id {67ff436c-ee93-483d-b694-d661063e6094}
   Property ModuleName: Id {eaa28a82-9f48-4672-adf0-02d762f98fa4}
   Get Get: Id {707fcee6-e5c4-4696-bdaf-64e6746ac511}
   Set Set: Id {29b514cf-0e85-455d-8f6d-dab417f76dd9}
   Property ParentResponse_Critical: Id {e581ea96-71f5-4214-b84f-fe40e4f439cd}
   Get Get: Id {cefd4a2e-0e84-4639-9399-50e5f85ba282}
   Set Set: Id {e602a147-21af-4f8b-a470-d7705d06bb99}
   Property ParentResponse_Error: Id {ea6cabed-35e0-4e31-9143-22fb00f7f237}
   Get Get: Id {90c102a5-e379-46b1-a6bc-51993d4e776d}
   Set Set: Id {2b602e0a-dc18-46ca-9ee2-e372c9159ca6}
   Property ParentResponse_Warning: Id {f50e684b-4ba8-413b-b162-40d548267b62}
   Get Get: Id {1eea4731-deef-4fce-9bd2-ce11f2ae2bde}
   Set Set: Id {d1e3f831-5a96-4cc4-83f2-65eaf98ff870}
   Property ParentResponseDef: Id {52bb93cb-0d1e-408e-9ae3-7e72a40e31ae}
   Get Get: Id {af09bce5-c0c6-4b5d-8736-3bc955f63074}
   Set Set: Id {1563a3c2-6b30-418c-b3a8-c6d3cce9d9ec}
   Method Resetting: Id {3807e2e0-6258-4c91-9f18-5b08f4f71847}
   Property SimulateAllChildren: Id {72dbc14c-7f4d-4f80-ac39-f560bdd6cdee}
   Get Get: Id {9993acbb-b83f-41c7-a0ae-e863eb1bca61}
   Set Set: Id {bbe57f06-302f-47bb-9f85-5cdcdfb0f46c}
   Method Starting: Id {ebd7ebd1-f8aa-4a46-a1fd-eef86be59683}
   Property State: Id {d1cab4fd-2e03-4869-8dbf-e461f1addf3b}
   Get Get: Id {650910fa-121e-4a38-96f8-196357ee8ede}
   Property StateCommand: Id {8c083f47-18a1-4a12-9399-91d5f5b4de80}
   Set Set: Id {7f7322f3-af6d-41b7-85ea-2b838219d81f}
   Method StateComplete: Id {0144eb9f-b619-4f85-a817-32c0b59111cc}
   Method StateControl: Id {adcfbb77-01ec-46bc-88f1-3c657cafd028}
   Method StopControlled: Id {6102a8b6-63d1-4349-9c91-23d23a740d56}
   Method StopImmediate: Id {4be9d206-4609-4609-8610-fb627d300ed2}
   Method Stopped: Id {6cf7e365-1763-4f32-a071-b4d38aa6475f}
   Method Stopping: Id {68934782-9f57-4361-9c27-3ced6fc0b6f9}
   Method SubModuleMonitor: Id {fe040716-db60-48a3-be9e-6ef7732045a6}
   Method SuspendControlled: Id {bf848d00-2f91-43a0-ba84-c03257f1e693}
   Method Suspended: Id {15a0521e-d09e-48c7-a5fb-e09a5fcfb990}
   Method SuspendImmediate: Id {541bc486-86e8-4c04-9fa3-e6a7ca36c7a0}
   Method Suspending: Id {9bd4e4e9-27b1-45dc-a32e-d60e4d2d284c}
   Property TargetProductionRate: Id {b514bd56-7d2e-4139-b530-8a3715ebc3bb}
   Get Get: Id {4bb69779-00b1-4880-914d-9920d90f543a}
   Set Set: Id {d78ceec9-4918-43fe-8cb1-bc0dc7830d6c}
   Method Undefined: Id {e1721cba-4da3-43ce-991b-54764c6d098b}
   Method Unholding: Id {d2ff920f-b2b8-44a1-a393-a69ebe202c6f}
   Method Unsuspending: Id {4c1e1471-15af-4f3d-8afa-3204208e7981}
   Method VISUCommunication: Id {566912f7-1ca8-4177-b0b8-f5f68d6072ff} *)
